FUNCTION invFrame : ST_Frame
VAR_INPUT
	i_frame :ST_Frame;
END_VAR
VAR
	invPos :Vec3d;
END_VAR

matTranspose(i_frame.m_rot, invFrame.m_rot);
vecMultiNum(i_frame.m_pos, -1, invPos);
matMultiVec(invFrame.m_rot, invPos, invFrame.m_pos);

END_FUNCTION

(* stored: Version 1.1.0.1, ProductVersion 3.1.4024.12
   POU invFrame: Id {e267f179-1cb3-4e2a-898f-03f4afe668ea}, SpecialFunc None *)
